// TIA Portal V20 export
DATA_BLOCK "BK25"   // DB273
// stored: MemoryReserve 100
   VAR
      "X10-1.JR WINDER REAR Y-AXIS LIMIT SENSOR(-)" : Bool := TRUE;
      "X10-2.JR WINDER REAR Y-AXIS HOME SENSOR" : Bool := FALSE;
      "X12-1.JR WINDER REAR Y-AXIS LIMIT SENSOR(+)" : Bool := TRUE;
      "X12-2.SPARE" : Bool := FALSE;
      "X14-1.JR WINDER FRONT Y-AXIS LIMIT SENSOR(-)" : Bool := TRUE;
      "X14-2.JR WINDER FRONT Y-AXIS HOME SENSOR" : Bool := TRUE;
      "X16-1.JR WINDER FRONT Y-AXIS LIMIT SENSOR(+)" : Bool := TRUE;
      "X16-2.SPARE" : Bool := FALSE;
   END_VAR
BEGIN
END_DATA_BLOCK
